FUNCTION_BLOCK AX_RS (* Event-driven bistable *)
  (* Standard: 61499-1 Annex A; Description: Copyright (c) 2017 fortiss GmbH, HR Agrartechnik GmbH This program and the accompanying materials are made available under the terms of the Eclipse Public License 2.0 which is available at https://www.eclipse.org/legal/epl-2.0/ SPDX-License-Identifier: EPL-2.0 *)
  (* Version 3.0, 2025-04-14, Patrick Aigner, changed package *)
  (* Version 1.0, 2017-09-22, Alois Zoitl, fortiss GmbH, initial API and implementation and/or initial documentation *)
  PACKAGE adapter::events::unidirectional;
  IMPORT eclipse4diac::core::TypeHash;
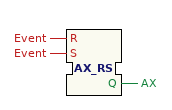
  EVENT_INPUT
    R; (* Reset output Q *)
    S; (* Set output Q *)
  END_EVENT
  PLUGS
    Q : adapter::types::unidirectional::AX; (* value of flip flop *)
  END_PLUGS
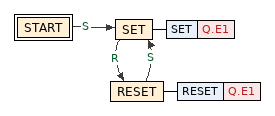
  EC_STATES
    START; (* Initial State *)
    SET : SET -> Q.E1;
    RESET : RESET -> Q.E1;
  END_STATES
  EC_TRANSITIONS
    START TO SET := S;
    SET TO RESET := R;
    RESET TO SET := S;
  END_TRANSITIONS
  ALGORITHM SET IN ST:
Q.D1 := TRUE;
  END_ALGORITHM
  ALGORITHM RESET IN ST:
Q.D1 := FALSE;
  END_ALGORITHM
END_FUNCTION_BLOCK
